{attribute addProperty BoxType "EK1122-0000-0018"}
{attribute addProperty Id "Beckhoff_EKx9xxsub_EK1100EK1100_179A0949162A_0001_EK1960_0000_0019EK1960_D284ECC656470.5A_0002_EK1960_0000_0021EK1960_858568AC53266.5A_0003_EK1960_0008_0019EK1960_D284ECC656470.5A_0004_EK1960_0008_0021EK1960_858568AC53266.5A_0005_EK1960_2600_0019EK1960_48A2E24356470.5A_0006_EK1960_2600_0021EK1960_3617E9AF56470.5A_0007_EK1960_2608_0019EK1960_48A2E24356470.5A_0008_EK1960_2608_0021EK1960_3617E9AF56470.5"}
{attribute addProperty CRC "429494437"}
{attribute addProperty SizeInBites "4464"}
{attribute addProperty SizeInBytes "558"}
TYPE Beckhoff_EKx9xxEK1122_199990A5 EXTENDS EK1122_179A0949 :
STRUCT
	{attribute addProperty Name "Beckhoff_EKx9xxsub_EK1100"}
	Beckhoff_EKx9xxsub_EK1100 : EK1100_179A0949;
	{attribute addProperty Name "A_0001_EK1960_0000_0019"}
	A_0001_EK1960_0000_0019 : EK1960_D284ECC6;
	{attribute addProperty Name "A_0002_EK1960_0000_0021"}
	A_0002_EK1960_0000_0021 : EK1960_858568AC;
	{attribute addProperty Name "A_0003_EK1960_0008_0019"}
	A_0003_EK1960_0008_0019 : EK1960_D284ECC6;
	{attribute addProperty Name "A_0004_EK1960_0008_0021"}
	A_0004_EK1960_0008_0021 : EK1960_858568AC;
	{attribute addProperty Name "A_0005_EK1960_2600_0019"}
	A_0005_EK1960_2600_0019 : EK1960_48A2E243;
	{attribute addProperty Name "A_0006_EK1960_2600_0021"}
	A_0006_EK1960_2600_0021 : EK1960_3617E9AF;
	{attribute addProperty Name "A_0007_EK1960_2608_0019"}
	A_0007_EK1960_2608_0019 : EK1960_48A2E243;
	{attribute addProperty Name "A_0008_EK1960_2608_0021"}
	A_0008_EK1960_2608_0021 : EK1960_3617E9AF;
END_STRUCT
END_TYPE

(* stored: Version 1.2.0.0, ProductVersion 3.1.4024.9
   DUT Beckhoff_EKx9xxEK1122_199990A5: Id {fb4e19bd-0f14-4291-94e7-324d0008312f} *)
